Universal Robots PolyScope program: easy_move.urp

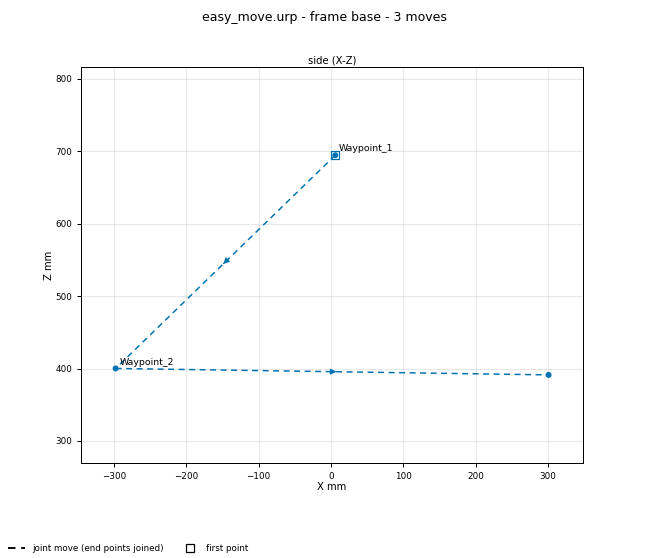
[picture p0: tool path of easy_move.urp in frame base, 3 of 3 moves have a stored position in this frame; points joined in program order, loops and branches not executed]
Program easy_move (installation=default directory=/programs/MW-UR createdIn=5.14.5 lastSavedIn=5.14.5 robotSerialNumber=20195300809)
Calibrated DH parameters: a=[-0.000085, -0.20076, -0.212369, 0.000121, -0.000118, 0]; d=[0.15185, -26.306375, 24.753047, 1.684739, 0.085386, 0.092088]; alpha=[1.572149, -0.00522, -0.011864, 1.571339, -1.571085, 0]; deltaTheta=[0, 0.599885, -0.513355, -0.086555, 0.000006, 0]
InitVariablesNode
Robot Program (runOnlyOnce=false)
  MoveJ speed 20 deg/s, acceleration 80 deg/s^2 (useActiveTCP=true) feature=Base
    Waypoint Waypoint_1: TCP in base x=5.909 y=-372.701 z=694.671 mm, rx=-0.0178 ry=2.2102 rz=-2.2165 rad; joints [-0.001, -89.998, 0, -90.002, -0.003, 0.003] deg; TCP offset x=0 y=0 z=150 mm, rx=0 ry=0 rz=0 rad
    Waypoint Waypoint_2: TCP in base x=-297.469 y=-374.476 z=400.116 mm, rx=1.1971 ry=1.2007 rz=-1.2133 rad; joints [0, -90.001, 89.999, -90.001, 0.002, 0.004] deg
    Waypoint Waypoint_3: TCP in base x=300.539 y=-371.898 z=391.229 mm, rx=1.221 ry=-1.2141 rz=1.2084 rad; joints [0.003, -89.999, -90.001, -89.997, 0.006, 0] deg
